RoboDK station: kr30 cnc 090919 2.rdk

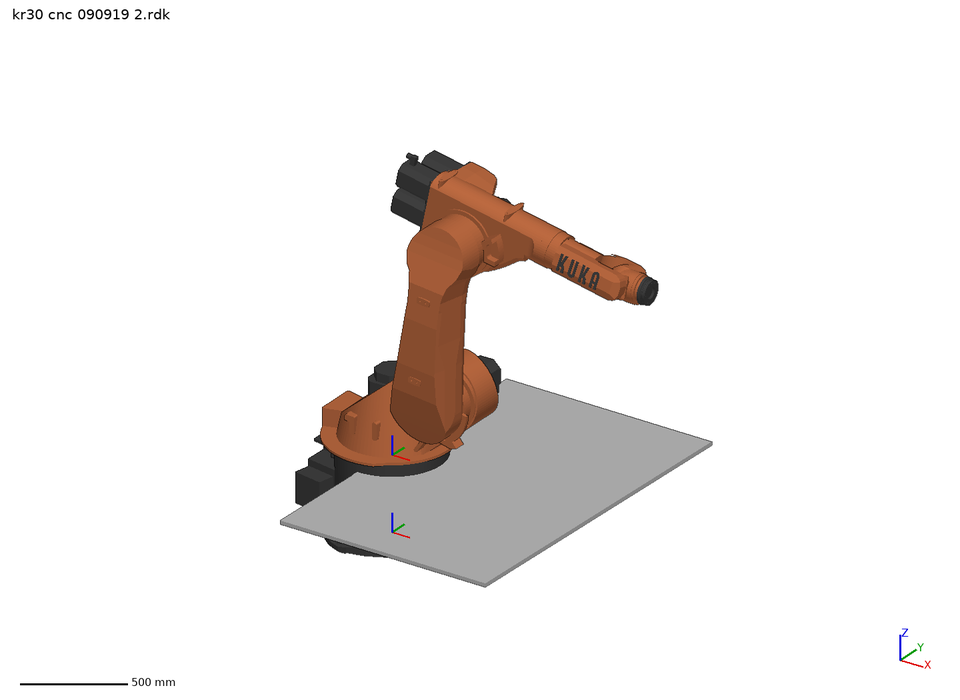
[picture v0: the station drawn from its stored meshes, robots at their saved joint values, targets as dots, program paths as lines]
Station kr30 cnc 090919 2. Poses are relative to the parent item; angles as X-Y-Z fixed-axis rotations.
  - frame KUKA KR 30 HA Base at (0, 0, 0) mm
    - robot KUKA KR 30 HA: 6 axes, payload 30 kg, reach 2033 mm, repeatability 0.05 mm, weight 665 kg
        modified DH rows (alpha deg, a mm, theta deg, d mm): 0, 0, 0, 815; -90, 350, 0, 0; 0, 850, -90, 0; -90, 145, 0, 820; 90, 0, 0, 0; -90, 0, 180, 170
        joint limits [-185, -135, -120, -350, -119, -350] to [185, 35, 158, 350, 119, 350]; home [0, -90, 90, 0, 0, 0]; saved at [-1.284, -83.635, 95.067, -345.51, -8.443, 347.45]
      - tool Angle Grinder (center shaft), TCP at (165.36, 24.52, 122.34) mm, geometry from KUKA KR 30 HA
    - frame Tabletop at (0, 0, 400) mm
      - object kr30 tabletop mm at (1160, -900, 0) mm, rotated rx 0 ry 0 rz 90 deg, size 1839.9 x 1168.4 x 19 mm, geometry from kr30 tabletop mm.stl
